{attribute 'qualified_only'}
VAR_GLOBAL CONSTANT
    const145_01Y : AxisLinMotConst_t := (POS_MIN := -5, POS_MAX := 200, VELO_MAX := 1000, VELO_MANU := 50);
    const145_02Z : AxisLinMotConst_t := (POS_MIN := -5, POS_MAX := 150, VELO_MAX := 1000, VELO_MANU := 50);
    const145_10W : AxisLinMotConst_t := (POS_MIN := 0, POS_MAX := 360, VELO_MAX := 360, VELO_MANU := 50);

END_VAR
VAR_GLOBAL
    axis145_01Y : AxisLinMot_t;
    axis145_02Z : AxisLinMot_t;
    axis145_10W : AxisLinMot_t;
END_VAR
VAR_GLOBAL RETAIN
    // Recipe values are managed elsewhere
END_VAR

(* stored: Version 1.1.0.1, ProductVersion 3.1.4024.6
   GVL ST145_Axis: Id {9d19c34b-b097-4509-8aa0-2c316c9c6fdc} *)
